// TIA Portal project "2026_05_08_Ciclio_A+_B+_T_A-_B-" (V15)

(* hardware
DEVICE "S7-1200 station_1"  S7-1200 Station
   slot 0: "Telaio di montaggio_0"  S7-1200 Rack  Rack  V1.0
   slot 1: "PLC_1"  CPU 1215C DC/DC/DC  6ES7 215-1AG40-0XB0  V4.2
*)

// ===== PLC "PLC_1"  CPU 1215C DC/DC/DC =====

VAR_GLOBAL   // PLC tag table "Tabella delle variabili standard"
   "System_Byte" AT %MB1 : Byte;
   "FirstScan" AT %M1.0 : Bool;
   "DiagStatusUpdate" AT %M1.1 : Bool;
   "AlwaysTRUE" AT %M1.2 : Bool;
   "AlwaysFALSE" AT %M1.3 : Bool;
   "Clock_Byte" AT %MB0 : Byte;
   "Clock_10Hz" AT %M0.0 : Bool;
   "Clock_5Hz" AT %M0.1 : Bool;
   "Clock_2.5Hz" AT %M0.2 : Bool;
   "Clock_2Hz" AT %M0.3 : Bool;
   "Clock_1.25Hz" AT %M0.4 : Bool;
   "Clock_1Hz" AT %M0.5 : Bool;
   "Clock_0.625Hz" AT %M0.6 : Bool;
   "Clock_0.5Hz" AT %M0.7 : Bool;
   "P_START" AT %I0.0 : Bool;
   "P_STOP" AT %I0.1 : Bool;
   "FC_A0" AT %I0.2 : Bool;
   "FC_A1" AT %I0.3 : Bool;
   "FC_B0" AT %I0.4 : Bool;
   "FC_B1" AT %I0.5 : Bool;
   "K" AT %M100.0 : Bool;
   "A+" AT %Q0.0 : Bool;
   "A-" AT %Q0.1 : Bool;
   "B+" AT %Q0.2 : Bool;
   "B-" AT %Q0.3 : Bool;
END_VAR

// folder: System blocks/Program resources

DATA_BLOCK "IEC_Timer_0_DB"   // DB1
{ S7_Optimized_Access := 'TRUE' }
AUTHOR : Simatic
FAMILY : IEC
NAME : IEC_TMR
VERSION : 1.0
// stored: InstanceOfName IEC_TIMER
"IEC_TIMER"
BEGIN
END_DATA_BLOCK

DATA_BLOCK "IEC_Timer_0_DB_1"   // DB2
{ S7_Optimized_Access := 'TRUE' }
AUTHOR : Simatic
FAMILY : IEC
NAME : IEC_TMR
VERSION : 1.0
// stored: InstanceOfName IEC_TIMER
"IEC_TIMER"
BEGIN
END_DATA_BLOCK

// folder: (top level)

ORGANIZATION_BLOCK "Main"   // OB1, LAD, ProgramCycle
TITLE = "Main Program Sweep (Cycle)"
{ S7_Optimized_Access := 'TRUE' }
VERSION : 0.1
   VAR_INPUT
      Initial_Call : Bool;   // Initial call of this OB
      Remanence : Bool;   // =True, if remanent data are available
   END_VAR
BEGIN

REGION Network 1: Enable
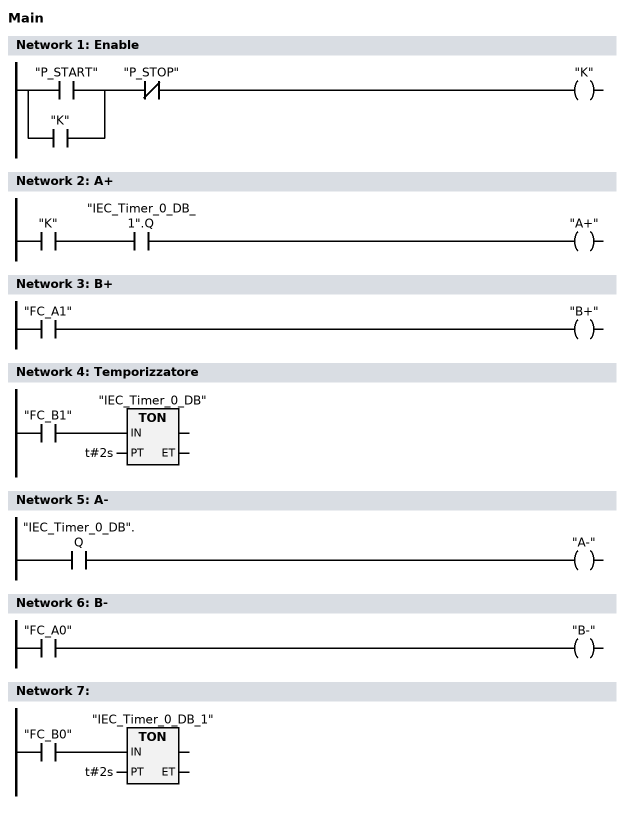
   RUNG wire#powerrail
      Contact( "P_START" )
      wire#w1
      I_Contact( "P_STOP" )
      Coil( "K" )
   END_RUNG
   RUNG wire#powerrail
      Contact( "K" )
   END_RUNG wire#w1
   // the same network as SCL:
   "K" := ("P_START" OR "K") AND NOT "P_STOP";
END_REGION

REGION Network 2: A+
   RUNG wire#powerrail
      Contact( "K" )
      Contact( "IEC_Timer_0_DB_1".Q )
      Coil( "A+" )
   END_RUNG
   // the same network as SCL:
   "A+" := "K" AND "IEC_Timer_0_DB_1".Q;
END_REGION

REGION Network 3: B+
   RUNG wire#powerrail
      Contact( "FC_A1" )
      Coil( "B+" )
   END_RUNG
   // the same network as SCL:
   "B+" := "FC_A1";
END_REGION

REGION Network 4: Temporizzatore
   "IEC_Timer_0_DB".TON(IN := "FC_B1", PT := t#2s);
END_REGION

REGION Network 5: A-
   RUNG wire#powerrail
      Contact( "IEC_Timer_0_DB".Q )
      Coil( "A-" )
   END_RUNG
   // the same network as SCL:
   "A-" := "IEC_Timer_0_DB".Q;
END_REGION

REGION Network 6: B-
   RUNG wire#powerrail
      Contact( "FC_A0" )
      Coil( "B-" )
   END_RUNG
   // the same network as SCL:
   "B-" := "FC_A0";
END_REGION

REGION Network 7
   "IEC_Timer_0_DB_1".TON(IN := "FC_B0", PT := t#2s);
END_REGION
END_ORGANIZATION_BLOCK